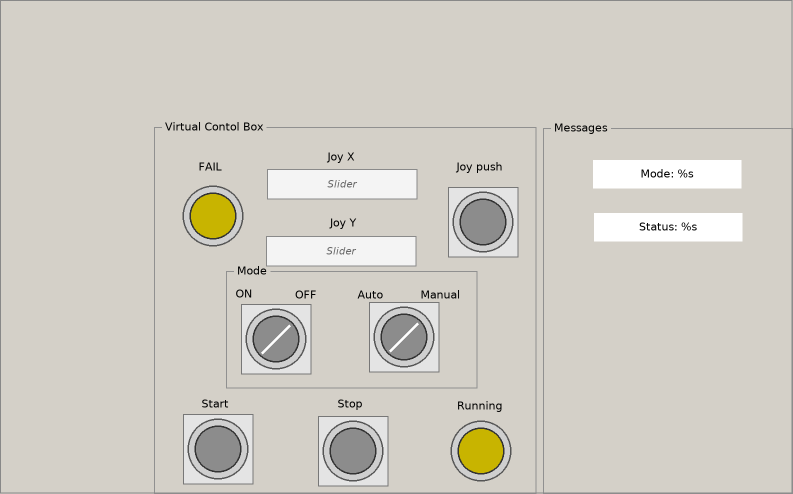
VISUALIZATION Visualization_1  // 793x494
    GroupBox (154,119 382x375), "Virtual Contol Box"
        GroupBox (72,144 251x125), "Mode"
            Label (56,17 48x30), "OFF"
            Label (0,16 36x30), "ON"
            RotarySwitch (143,39 70x70), variable: GVL_HMI.st_box_param.bAuto, behaviour: TOGGLE, style: Switch-RotarySwitch-Gray
            Label (105,17 79x30), "Auto"
            RotarySwitch (15,41 70x70), variable: GVL_HMI.st_box_param.bReady, behaviour: TOGGLE, style: Switch-RotarySwitch-Gray
        PushSwitchLed (29,295 70x70), variable: GVL_HMI.st_box_param.bStarting, behaviour: TAP, style: Switch-PushSwitchLed-Gray
        PushSwitchLed (164,297 70x70), variable: GVL_HMI.st_box_param.bStopping, behaviour: TAP, style: Switch-PushSwitchLed-Gray
        Label (167,270 58x30), "Stop"
        Label (247,161 79x30), "Manual"
        Label (30,270 62x30), "Start"
        Slider (113,50 150x30), variable: GVL_HMI.st_box_param.fJoy_X, scale 0..32767
        Label (112,23 150x30), "Joy X"
        Slider (112,117 150x30), variable: GVL_HMI.st_box_param.fJoy_Y, scale 0..32767
        Label (114,89 150x30), "Joy Y"
        PushSwitchLed (294,68 70x70), variable: GVL_HMI.st_box_param.bJoyPush, behaviour: TAP, style: Switch-PushSwitchLed-Gray
        Lamp1 (292,297 70x70), variable: GVL_HMI.st_box_param.bRunning, style: Lamp-Lamp1-Yellow
        Label (297,272 58x30), "Running"
        Label (293,33 65x30), "Joy push"
        Lamp1 (24,62 70x70), variable: GVL_HMI.st_box_param.bFault, style: Lamp-Lamp1-Yellow
        Label (27,33 58x30), "FAIL"
    GroupBox (543,120 250x374), "Messages"
        Textfield (50,92 150x30), "Status: %s", text variable: GVL_HMI.eStatus
        Textfield (49,39 150x30), "Mode: %s", text variable: GVL_HMI.eMode
END_VISUALIZATION

(* stored: Version 1.1.0.1, ProductVersion 3.1.4024.12
   Visu Visualization_1: Id {e6407bed-d73d-4f13-b1ea-fe75486f8fd1} *)
